(* Logix 5000 project; controller CLP_AB vendor 1 type 14 code 79 rev 17.4; software revision 17.01 *)

TASK DeviceNet (continuous, watchdog 500 ms) : DeviceN
TASK Initialize_speed (event, rate 10 ms, priority 10, watchdog 500 ms) : Initialize_Data
TASK MainTask (periodic, rate 46.875 ms, priority 10, watchdog 500 ms) : Camera_Trigger

MODULES
   Local : vendor 1 type 14 code 79 (ICP 0, rev 17.4)
      DN : vendor 1 type 12 code 14 (ICP 2, rev 7.3, Output RPI 20 ms, Input RPI 20 ms)
      Ethernet : 1756-ENBT (Ethernet 192.168.0.4, ICP 3, rev 4.1)
         Camera_Sensor : ETHERNET-MODULE (Ethernet 192.168.0.3, rev 1.1, Output RPI 25 ms)   // Banner
      LocalSERCOS : vendor 1 type 16 code 14 (ICP 1, rev 17.2, MotionAsync RPI 25 ms, MotionEvent RPI 1000 ms, MotionSync RPI 2 ms)
         Drive : vendor 1 type 115 code 164 (SERCOS 1, rev 1.1)
END_MODULES

VAR_GLOBAL   (* controller tags *)
   BitTest1 : BOOL;
   BitTest2 : BOOL;
   botao : BOOL;
   dataInitialized : BOOL;
   dir_int : DINT;
   direction : BOOL;
   drive_axis : AXIS_SERVO_DRIVE;
   Emanuel : BOOL;
   encoder : AXIS_SERVO_DRIVE;
   IterationChange : ALIAS FOR Camera_Sensor:I.Data[6].0;
   IterationChanged : BOOL;
   IterationCount : DINT;
   lastIterationCount : DINT;
   MAH_0 : MOTION_INSTRUCTION;
   MAJ_0 : MOTION_INSTRUCTION := (FLAGS := 33554432);
   MAJ_1 : MOTION_INSTRUCTION := (FLAGS := 33554432);
   MAJ_2 : MOTION_INSTRUCTION;
   MAS_0 : MOTION_INSTRUCTION;
   MAS_1 : MOTION_INSTRUCTION := (FLAGS := 33554432);
   MAS_2 : MOTION_INSTRUCTION;
   MGroup : MOTION_GROUP;
   MSF_0 : MOTION_INSTRUCTION;
   MSO_0 : MOTION_INSTRUCTION;
   MSO_1 : MOTION_INSTRUCTION := (FLAGS := -1610612736, EN := 1, DN := 1, STATE := 1);
   OutTest1 : BOOL;
   OutTest2 : BOOL;
   position : ALIAS FOR Camera_Sensor:I.Data[16];
   Ready : ALIAS FOR Camera_Sensor:I.Data[0].4;
   speed : REAL[342];
   speedRate : REAL;
   timer_1 : TIMER := (PRE := 500);
   Trigger_ACK : ALIAS FOR Camera_Sensor:I.Data[0].16;
   trigger_off : TIMER := (PRE := 10);
   trigger_on : TIMER := (PRE := 10);
END_VAR

PROGRAM Camera_Trigger   (* main routine TriggerMain *)
// Trigger
VAR
   Trigger : ALIAS FOR Camera_Sensor:O.Data[0].0;
END_VAR

ROUTINE TriggerMain   (* ladder *)
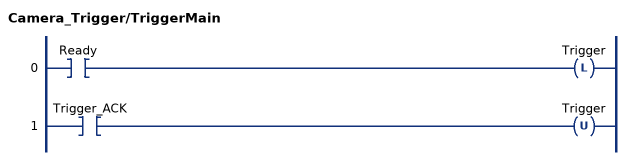
   0: XIC(Ready)OTL(Trigger);
   1: XIC(Trigger_ACK)OTU(Trigger);
END_ROUTINE
END_PROGRAM

PROGRAM Controle   (* main routine malhaAberta *)
VAR
   direcMove : DINT;
   k : DINT;
   timervel : FBD_TIMER;
END_VAR

ROUTINE ControleMain   (* structured text *)
   COP(Camera_Sensor:I.Data[6],IterationCount,32);
   if IterationCount > lastIterationCount then
   	/*Aqui vai o nosso controlador*/
   	if position > 205.0 then
   		speedRate:=.2;
   		direcMove:=1;
   	elsif position < 195.0 then
   		speedRate:=.2;
   		direcMove:=0;
   	else
   		speedRate:=0;
   		MAS(drive_axis,MAS_1,0,0,100,1,0,100,1);
   	end_if;
   	MAJ(drive_axis,MAJ_1,direcMove,speedRate,0,50.0,1,50.0,1,0,50.0,50.0,1,0,0);
   	COP(Camera_Sensor:I.Data[6],lastIterationCount,32);
   end_if;
END_ROUTINE

ROUTINE malhaAberta   (* structured text *)
   // k is the index of the speed vector
   if dataInitialized AND k < 85 then
   	MAJ(drive_axis,MAJ_1,0,speed[k],0,50.0,1,50.0,1,0,50.0,50.0,1,0,0);
   	k:=k + 1;
   end_if;
   
   if k >= 85 then
   	MAS(drive_axis,MAS_1,0,0,100,1,0,100,1);
   	if MAS_1.DN then
   		MSF(drive_axis,MSF_0);
   	end_if;
   end_if;
END_ROUTINE

ROUTINE VeloMain   (* structured text *)
   COP(Camera_Sensor:I.Data[6],IterationCount,32);
   /*MAJ(drive_axis,MAJ_1,0,0.5,0,50.0,1,50.0,1,0,50.0,50.0,1,0,0);
   timervel.TimerEnable:=1;
   TONR(timervel);
   MAS(drive_axis,MAS_1,All,0,100,1,0,100,1);
   MSF(drive_axis,MSF_0);
   */
   	//MSO(drive_axis,MSO_1);
   	timervel.PRE:=20000;
   	if (MSO_1.EN AND timervel.ACC < 20000) then
   		if (NOT timervel.DN) then
   			timervel.TimerEnable:=1;
   			MAJ(drive_axis,MAJ_1,0,0.2,0,50.0,1,50.0,1,0,50.0,50.0,1,0,0);
   			TONR(timervel);
   		end_if;
   	end_if;
   	if (timervel.DN) then
   		MAS(drive_axis,MAS_1,All,0,100,1,0,100,1);
   	end_if;
   	if (MAS_1.EN) then
   		MSF(drive_axis,MSF_0);
   	end_if;
   
END_ROUTINE
END_PROGRAM

PROGRAM Controle1   (* main routine VeloMain *)
VAR
   direcMove : DINT;
   timervel : FBD_TIMER;
END_VAR

ROUTINE ControleMain   (* structured text *)
   COP(Camera_Sensor:I.Data[6],IterationCount,32);
   if IterationCount > lastIterationCount then
   	/*Aqui vai o nosso controlador*/
   	if position > 205.0 then
   		speedRate:=.2;
   		direcMove:=1;
   	elsif position < 195.0 then
   		speedRate:=.2;
   		direcMove:=0;
   	else
   		speedRate:=0;
   		MAS(drive_axis,MAS_1,0,0,100,1,0,100,1);
   	end_if;
   	MAJ(drive_axis,MAJ_1,direcMove,speedRate,0,50.0,1,50.0,1,0,50.0,50.0,1,0,0);
   	COP(Camera_Sensor:I.Data[6],lastIterationCount,32);
   end_if;
END_ROUTINE

ROUTINE VeloMain   (* structured text *)
   COP(Camera_Sensor:I.Data[6],IterationCount,32);
   /*MAJ(drive_axis,MAJ_1,0,0.5,0,50.0,1,50.0,1,0,50.0,50.0,1,0,0);
   timervel.TimerEnable:=1;
   TONR(timervel);
   MAS(drive_axis,MAS_1,All,0,100,1,0,100,1);
   MSF(drive_axis,MSF_0);
   */
   	//MSO(drive_axis,MSO_1);
   	timervel.PRE:=20000;
   	if (MSO_1.EN AND timervel.ACC < 20000) then
   		if (NOT timervel.DN) then
   			timervel.TimerEnable:=1;
   			MAJ(drive_axis,MAJ_1,0,0.2,0,50.0,1,50.0,1,0,50.0,50.0,1,0,0);
   			TONR(timervel);
   		end_if;
   	end_if;
   	if (timervel.DN) then
   		MAS(drive_axis,MAS_1,All,0,100,1,0,100,1);
   	end_if;
   	if (MAS_1.EN) then
   		MSF(drive_axis,MSF_0);
   	end_if;
   
END_ROUTINE
END_PROGRAM

PROGRAM DeviceN   (* main routine InitDNetST *)

ROUTINE InitDNetST   (* structured text *)
   Local:2:O.CommandRegister.Run [:=] 1;
   if NOT dataInitialized then
   	EVENT(Initialize_speed);
   end_if;
   
END_ROUTINE
END_PROGRAM

PROGRAM Initialize_Data   (* main routine Init *)

ROUTINE Init   (* structured text *)
   /* Universidade de Brasilia
   Trabalho de Graduacao em Engenharia Mecatronica
   Alunos:
   Ataias Pereira Reis 10/0093817
   Emanuel Pereira Barroso Neto 11/0115716
   This code must be executed only once. */
   
   MSO(drive_axis,MSO_1);
   
   speed[0] := 0.0;
   speed[1] := 0.0;
   speed[2] := 0.0;
   speed[3] := 0.0;
   speed[4] := 0.0;
   speed[5] := 0.0;
   speed[6] := 0.0;
   speed[7] := 0.0;
   speed[8] := 0.0;
   speed[9] := 0.0;
   speed[10] := 0.0;
   speed[11] := 0.0;
   speed[12] := 0.0;
   speed[13] := 0.0;
   speed[14] := 0.0;
   speed[15] := 0.0;
   speed[16] := 0.0;
   speed[17] := 0.0;
   speed[18] := -0.0692113524459;
   speed[19] := 0.314942000684;
   speed[20] := 1.64847179452;
   speed[21] := 3.06203932423;
   speed[22] := 3.88556305076;
   speed[23] := 4.25984881416;
   speed[24] := 4.24772217569;
   speed[25] := 3.9166637819;
   speed[26] := 3.35019221407;
   speed[27] := 2.64853848716;
   speed[28] := 1.92086693496;
   speed[29] := 1.27214274157;
   speed[30] := 0.788466188462;
   speed[31] := 0.524290908189;
   speed[32] := 0.493490156489;
   speed[33] := 0.694837969193;
   speed[34] := 0.822419246039;
   speed[35] := 0.418206857379;
   speed[36] := 0.0262247526643;
   speed[37] := 0.230482402967;
   speed[38] := 0.789536874806;
   speed[39] := 1.48057490162;
   speed[40] := 2.15097967763;
   speed[41] := 2.69969451667;
   speed[42] := 3.0612889055;
   speed[43] := 3.19935866684;
   speed[44] := 3.10564873155;
   speed[45] := 2.7984308071;
   speed[46] := 2.32194132411;
   speed[47] := 1.78925311378;
   speed[48] := 1.23475193349;
   speed[49] := 0.680977178876;
   speed[50] := 0.269581981875;
   speed[51] := 0.0735006589406;
   speed[52] := 0.0;
   speed[53] := -0.0411084579085;
   speed[54] := -0.0752386045019;
   speed[55] := -0.0939490510793;
   speed[56] := -0.0958419020537;
   speed[57] := -0.0879379646741;
   speed[58] := -0.0665110466718;
   speed[59] := -0.0340396907113;
   speed[60] := 0.0;
   speed[61] := 0.0116207365686;
   speed[62] := 0.0239437089848;
   speed[63] := 0.0232352765649;
   speed[64] := 0.0;
   speed[65] := 0.0;
   speed[66] := 0.0;
   speed[67] := 0.0;
   speed[68] := 0.0;
   speed[69] := 0.0;
   speed[70] := 0.0;
   speed[71] := 0.0;
   speed[72] := 0.0;
   speed[73] := 0.0;
   speed[74] := 0.0;
   speed[75] := 0.0;
   speed[76] := 0.0;
   speed[77] := 0.0;
   speed[78] := 0.0;
   speed[79] := 0.0;
   speed[80] := 0.0;
   speed[81] := 0.0;
   speed[82] := 0.0;
   speed[83] := 0.0;
   speed[84] := 0.0;
   speed[85] := 0.0;
   
   dataInitialized := 1;
   
END_ROUTINE
END_PROGRAM

PROGRAM MainProgram   (* main routine MainRoutineST *)

ROUTINE MainRoutine   (* ladder *)
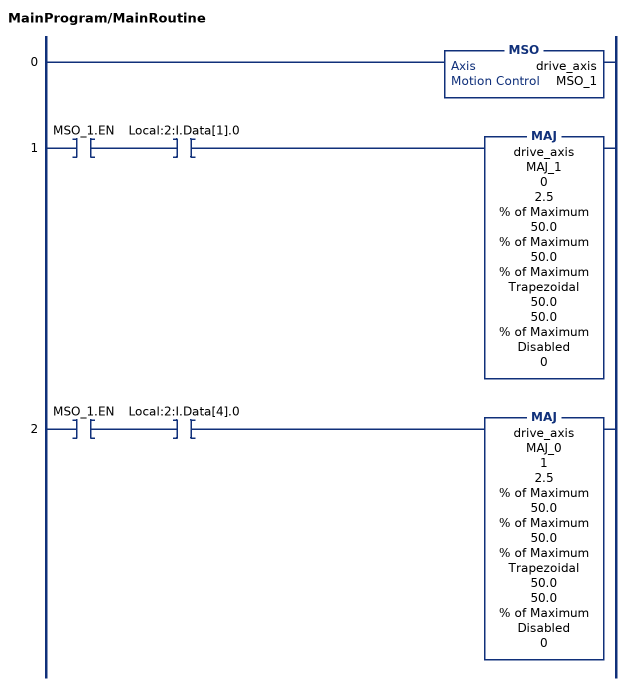
   0: MSO(drive_axis,MSO_1);
   1: XIC(MSO_1.EN)XIC(Local:2:I.Data[1].0)MAJ(drive_axis,MAJ_1,0,2.5,% of Maximum,50.0,% of Maximum,50.0,% of Maximum,Trapezoidal,50.0,50.0,% of Maximum,Disabled,0);
   2: XIC(MSO_1.EN)XIC(Local:2:I.Data[4].0)MAJ(drive_axis,MAJ_0,1,2.5,% of Maximum,50.0,% of Maximum,50.0,% of Maximum,Trapezoidal,50.0,50.0,% of Maximum,Disabled,0);
END_ROUTINE

ROUTINE MainRoutineST   (* structured text *)
   MSO(drive_axis,MSO_1);
   IF MSO_1.EN AND Local:2:I.Data[1].0 THEN
   	MAJ(drive_axis,MAJ_1,0,2.5,1,50.0,1,50.0,1,0,50.0,50.0,1,0,0);
   END_IF;
   IF MSO_1.EN AND Local:2:I.Data[4].0 THEN
   	MAJ(drive_axis,MAJ_0,1,2.5,1,50.0,1,50.0,1,0,50.0,50.0,1,0,0);
   END_IF;
END_ROUTINE
END_PROGRAM

PROGRAM Parada   (* main routine parada *)

ROUTINE parada   (* ladder *)
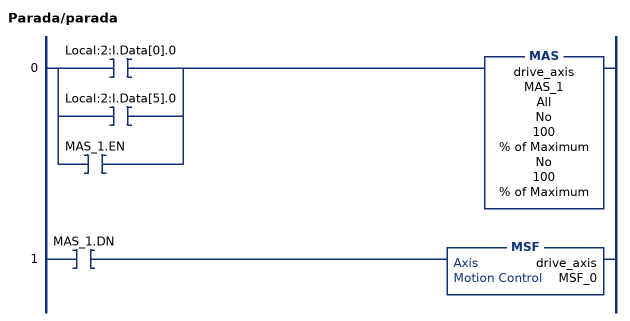
   0: [XIC(Local:2:I.Data[0].0) ,[XIC(Local:2:I.Data[5].0) ,XIC(MAS_1.EN) ] ]MAS(drive_axis,MAS_1,All,No,100,% of Maximum,No,100,% of Maximum);
   1: XIC(MAS_1.DN)MSF(drive_axis,MSF_0);
END_ROUTINE
END_PROGRAM
